PROGRAM PRG_Machine
VAR
	
	//empty recipe
	empty_recipe				:recipe;
	
	//debug
	after_debug_state					:INT :=0;

	
	Pusher :FB_Pusher;
	Compress: FB_Compress;
	Shield: FB_Shield;

	ZenonStart: NT_StartProcess;

	
	debug_counter: INT;
	tickcounter: INT;
	tickcounter2: INT;

	State: INT:= 0;
	state_old: INT:=0;
	StateNext: INT:= 0;
	
	SM_StepRequest: BOOL:=FALSE;
	singleStep: BOOL:=FALSE;
		
	Clamp_Security_Time: TIME := T#30S;
	ClampTimer: TON;
	//DwellTimer: TON;
	//SaveTickCounter: INT := 0;

	DatumTaught: BOOL;

	

	
	//stage
	stage_sh_push						:INT:=1;
	
END_VAR

VAR_OUTPUT

	rec_old		:recipe;
END_VAR

IF TRUE THEN
	debug_counter := debug_counter+1;
END_IF



qbCompressServoTorqueLimit := 1000;
qbPusherServoTorqueLimit := 1000;
qbShieldServoTorqueLimit := 1000;


//The state-machine
CASE State OF
	
0: //Copy config .txt file into machine settings
	


	//Zenon start process function call - appears to never generate errors
	
	//IF ZenonStart.Busy=FALSE THEN
	ZenonStart (
		NETID :=,
		//PATHSTR := 'Hard Disk\CP6606_Runtime\zenonRCE.exe', //'C:\PROGRAM Files\COPA-DATA\zenon 7.20 SP0\Zenrt32.exe',
		//DIRNAME := 'Hard Disk\CP6606_Runtime',  //'C:\Program Files\COPA-DATA\zenon 7.20 SP0',
		PATHSTR := 'Hard Disk\ZenonRunTime\zenonRCE.exe', //'C:\PROGRAM Files\COPA-DATA\zenon 7.20 SP0\Zenrt32.exe',
		DIRNAME := 'Hard Disk\ZenonRunTime',  //'C:\Program Files\COPA-DATA\zenon 7.20 SP0',
		COMNDLINE := '',
		START := TRUE,
		TMOUT := DEFAULT_ADS_TIMEOUT
		);
	StateNext := 10;



10: 
	qxEnableE_Stop := FALSE;
	tickcounter := 0;
	StateNext := 15;

15: //Check E-Stop relay is not set then Enable and initialise stuff - disable drive to clear errors

	

	//IF ixCabinetE_StopButtonOkay THEN
	qxEnableE_Stop := TRUE;
	StateNext := 20;
	//ELSE
	//	ResetLampController.State := SlowFlash;
	//END_IF
	
20: // Look for E-Stop button reset
	IF ixCabinetE_StopButtonOkay THEN
		//ResetLampController.State := steady;
		StateNext := 30;
	ELSE
		 
		ResetLampController.State := SlowFlash;
			
	END_IF
	
	//here
30: // Wait for operator to hit reset button
	
	IF ixE_StopRelayOkay THEN
		ResetLampController.State := off;
		StateNext := 40;
		tickcounter := 0;
	ELSE
		ResetLampController.State := steady;
		


	END_IF

40: // look for guard closed - disable drive to clear errors
	//sSystemStateMed := F_DisplayText("Guard Open",0);	
	//CurrentProcessState	:= F_DisplayText("not ready",0);	//Main Screen	

	
	IF NOT ixGuardOkay THEN
		ResetLampController.State := FastFlash;		
	ELSE
		ResetLampController.State := off;
		//sSystemStateMed := F_DisplayText("Initialising Axes",0);	
		tickcounter := 0;
		StateNext := 50;
	END_IF

50:
	IF ixGuardRelayOkay THEN
		statenext:=100;
	END_IF
	
100: // wait 2 scans for power supply to drive to stabilise
	tickcounter := tickcounter + 1;
	IF tickcounter >= 2 THEN
		tickcounter := 0;
		StateNext := 105;
	END_IF

105:
	IF NOT ixresetbutton THEN
		statenext:=110;
	END_IF	
	
110: // prepare for Servo motion - enable drive
//you are here!!!!!!!!!!!!!!!!!!!!!!!!!!!!
	//IF NOT ixResetButton THEN
		
		
	
	Shield._Enable();
	Pusher._Enable();
	Compress._Enable();
		
	tickcounter := tickcounter + 1;
	IF tickcounter >= 100 THEN
		tickcounter := 0;

		StateNext := 115;
	END_IF	
	//END_IF


	
115: 
	
	//IF Shield.HomeExecuted = FALSE OR Pusher.HomeExecuted = FALSE OR Compress.HomeExecuted = FALSE THEN
	IF language.english THEN
		Stage_Name := 'Beginning';
	ELSE
		Stage_Name := 'Início';
	END_IF
	Maintenance_Visibility:=TRUE;
	qxStartButtonLamp:=TRUE;
	IF (ixStartButton OR Step_Next OR ixStart_Button_Machine) THEN
		IF (parameter_violation = FALSE) THEN
			qxStartButtonLamp:=FALSE;
			StateNext := 116;
			Step_Next := FALSE;
			Clamp_Alarm:=FALSE;
			Maintenance_Visibility:=FALSE;
			stage_sh_push:=1;
			//Stage_Name := 'Homing and Offsetting';



		ELSE
			Step_Next:=FALSE;
		END_IF
	END_IF

	
116:
	IF (NOT ixstartbutton) AND NOT ixstart_button_machine THEN
		//general_offset_update();

		
		statenext:=117;
	END_IF
	
117:
	IF Compress.HomeExecuted=TRUE AND 
	   Shield.HomeExecuted = TRUE AND 
	   Pusher.HomeExecuted = TRUE AND
	   Pusher.OffsetExecuted = TRUE AND
	   Shield.OffsetExecuted = TRUE AND
	   Compress.OffsetExecuted = TRUE AND
	   Debug_Mode = FALSE THEN
	   
	   statenext:= 130;
	ELSE
		statenext:=120;
	END_IF
	
	Shield.Shield_param:=recipe_screen;
	Compress.Compress_Param := recipe_screen;
	Pusher.Pusher_Param := recipe_screen;
	//ELSE
	//	StateNext:=129;
	//	after_debug_state:=128;
	//END_IF
		
120: //you are here!!!!!!!!!!!!

	IF language.english THEN
		Stage_Name := 'Homing';
	ELSE
		Stage_Name := 'Ir para Início';
	END_IF
	IF Pusher.HomeExecuted = FALSE THEN 
		Pusher._Home();
	END_IF
	
	IF Compress.HomeExecuted = FALSE THEN
		Compress._Home();
	END_IF
	
	
	IF Compress.HomeExecuted AND Pusher.HomeExecuted THEN
		StateNext := 125;                //directly to end
		//Compress.HomeExecuted:=FALSE;
		//Pusher.HomeExecuted:=FALSE;
		
	END_IF
	
125:
	//random:='arda';
	IF Shield.HomeExecuted = FALSE THEN
		Shield._Home();
		
	ELSE
		StateNext := 129;
		IF language.english THEN
			Stage_Name := 'Homing done';
		ELSE
			Stage_Name := 'Ir para início concluído';
		END_IF
		after_debug_state :=127;
		//Shield.HomeExecuted := FALSE;
	END_IF

127:
	
	IF language.english THEN	
		Stage_Name := 'Offsetting';
	ELSE
		Stage_Name := 'Desviando';
	END_IF
	
	IF Compress.OffsetExecuted = FALSE THEN
		Compress.Offset(enable:=TRUE);
	END_IF
	
	IF Shield.OffsetExecuted = FALSE THEN
		Shield.Offset(enable:=TRUE);
	END_IF
	
	IF Pusher.OffsetExecuted = FALSE THEN
		Pusher.Offset(enable:=TRUE);
	END_IF
	
	IF Pusher.OffsetExecuted AND Shield.OffsetExecuted AND Compress.OffsetExecuted THEN
		Pusher.Offset(enable:=FALSE);
		Shield.Offset(enable:=FALSE);
		Compress.Offset(enable:=FALSE);
		
		rec_old:=Shield.Shield_Param;     //old values
		
		IF language.english THEN
			Stage_Name := 'Offsetting done';
		ELSE
			Stage_Name :='Desvio concluído';	
		END_IF
		
		Maintenance_Visibility := TRUE;
		qxStartButtonLamp:=TRUE;
		IF (ixStartButton OR Step_Next OR ixStart_Button_Machine) THEN
			IF (parameter_violation =FALSE) THEN
				qxStartButtonLamp:=FALSE;
				
				Shield.Shield_param:=recipe_screen;
				Compress.Compress_Param := recipe_screen;
				Pusher.Pusher_Param := recipe_screen;
			
				StateNext:=128;
				Step_Next:=FALSE;
				Maintenance_Visibility := FALSE;
			ELSE
				Step_Next:=FALSE;
			END_IF
		END_IF
	END_IF
	
128:	
	IF NOT ixstartbutton AND NOT ixstart_button_machine THEN
		statenext:=130;
	END_IF	

129: //debug	
	
	IF _debug(enable:=TRUE) THEN
		_debug(enable:=FALSE);
		statenext:=131;
	END_IF
		
130: //stage 1

	//IF ixstartbutton AND NOT ixstart_button_machine THEN
	IF language.english THEN
		Stage_Name := 'Compress Tobacco';
	ELSE
		Stage_Name := 'Comprimir Tabaco';
	END_IF
	
	IF qxClamp = FALSE THEN
		qxClamp:=TRUE;
		ClampTimer.IN:=TRUE;
		ClampTimer.PT:=Clamp_Security_Time;

	END_IF
	
	//IF Compress.Stage1Executed = FALSE THEN

	Compress._compress_tobacco(Enable:=TRUE);
	Compress.HomeExecuted:=FALSE;	
	
	IF Compress.axis_ready THEN	//Compress.Stage1Executed := FALSE;
		StateNext := 129;
		after_debug_state:=135;
		Compress._compress_tobacco(Enable:=FALSE);
		
		
		IF language.english THEN
			Stage_Name := 'Compress Tobacco done';
		ELSE
			Stage_Name := 'Comprimir tabaco concluído';
		END_IF
		
	END_IF
	//END_IF

131: //after_each_debug
	IF NOT ixStartButton AND NOT ixStart_Button_Machine THEN
	
		statenext:=after_debug_state;
	END_IF
135://stage2
	
	IF language.english THEN
		Stage_Name := concat('Shield-Pusher Stage ',INT_TO_STRING(stage_sh_push));
	ELSE
		Stage_Name := concat('Empurrador-proteção Estágio',INT_TO_STRING(stage_sh_push));
	END_IF
	
	Pusher.HomeExecuted:=FALSE;
	Shield.HomeExecuted:=FALSE;
		
	Pusher._absolute_move(Enable:=TRUE,Stage:=stage_sh_push);
	Shield._absolute_move(Enable:=TRUE,Stage:=stage_sh_push);
	IF pusher.axis_ready AND shield.axis_ready THEN	
		Statenext:= 129;
		IF stage_sh_push =6 THEN
			after_debug_state := 150;
			stage_sh_push:=0;
		ELSE
			after_debug_state := 135;
		END_IF
		Pusher._absolute_move(Enable:=FALSE,Stage:=stage_sh_push);
		Shield._absolute_move(Enable:=FALSE,Stage:=stage_sh_push);
		stage_sh_push:=stage_sh_push+1;
		
		IF language.english THEN
			Stage_Name:=concat(Stage_Name,' done');
		ELSE
			Stage_Name:=concat(Stage_Name,' concluído');
		END_IF
	END_IF	
	


150: //stage 5
	IF language.english THEN
		Stage_Name := 'Retract all';
	ELSE
		Stage_Name := 'Retrair tudo';
	END_IF
	//IF 	Shield._retract(Enable:=TRUE) AND Pusher._retract(Enable:=TRUE) AND Compress._retract(Enable:=TRRUE) THEN
	Pusher._Retract(enable:=TRUE);
	Shield._retract(enable:=TRUE);
	Compress._retract(enable:=TRUE);

	IF Compress.axis_ready AND Shield.Axis_ready AND Pusher.axis_ready THEN
		Pusher._Retract(enable:=FALSE);
		Shield._retract(enable:=FALSE);
		Compress._retract(enable:=FALSE);
		Statenext:=290;
		
		IF language.english THEN
			Stage_Name := 'Retract All Done';
		ELSE
			Stage_Name := 'Retrair tudo concluído';
		END_IF
	END_IF	

290:
	product_count:=product_count+1;
	statenext:=300;


300: //end
	
	Pusher.HomeExecuted:= TRUE;
	Shield.HomeExecuted:=TRUE;
	Compress.HomeExecuted:=TRUE;
	statenext:= 115;

	
1000: // overtorque
	
	//StartLoad := FALSE;
	
	tickcounter:=0;
	
	qxclamp:=FALSE;
	ClampTimer.IN:=FALSE;
	ClampTimer.PT:=Clamp_Security_Time;
	
	IF Pusher.PusherServo.xstopped AND Shield.ShieldServo.xstopped AND Compress.CompressServo.xstopped THEN
		Pusher._Reset();
		Shield._Reset();
		Compress._Reset();
		Statenext:=1005;
	END_IF

1005:
	
	IF tickcounter >1000 THEN
		statenext:=2000;
		tickcounter:=0;
	ELSE
		tickcounter:=tickcounter+1;
	END_IF

	
2000: // estop //overtorque
	
	tickcounter:= tickcounter+1;
	IF	tickcounter = 100 THEN
		tickcounter:=0;
		
		statenext:=15;
		overtorque_alarm:=FALSE;
	END_IF

2001: //guard
	tickcounter:= tickcounter+1;
	IF	tickcounter = 100 THEN
		tickcounter:=0;
		
		statenext:= 40;
		
	END_IF

2010: // clamp alarm
	
	tickcounter:= tickcounter+1;

	
	IF clamp_alarm THEN
		
		IF	tickcounter = 3000 THEN
			tickcounter:=0;
			statenext:=100;
			Clamp_Cooling := FALSE;
			Clamp_Alarm := FALSE;
		ELSE
			Clamp_Cooling := TRUE;
			
			IF Pusher.PusherServo.xstopped AND Shield.ShieldServo.xstopped AND Compress.CompressServo.xstopped THEN
				Pusher._Reset();
				Shield._Reset();
				Compress._Reset();
			END_IF
		END_IF
	END_IF 



2015://stop button
	tickcounter:= tickcounter+1;
	IF	tickcounter = 100 THEN
		tickcounter:=0;
		statenext:=100;
		
	ELSIF Pusher.PusherServo.xstopped AND Shield.ShieldServo.xstopped AND Compress.CompressServo.xstopped THEN
		Pusher._Reset();
		Shield._Reset();
		Compress._Reset();
		
	END_IF

2020: //force home

	IF shield.ShieldServo.xHalted AND pusher.pusherservo.xHalted AND compress.compressservo.xhalted THEN
		Pusher._soft_Reset();
		Shield._soft_Reset();
		Compress._soft_Reset();
		IF compress.offsetExecuted AND shield.Offsetexecuted AND pusher.offsetexecuted THEN
			statenext:=200;
		ELSE

			statenext:=210;
		END_IF
	END_IF

2030: //compress setting
	IF shield.ShieldServo.xHalted AND pusher.pusherservo.xHalted AND compress.compressservo.xhalted THEN
		Pusher._soft_Reset();
		Shield._soft_Reset();
		Compress._soft_Reset();
		
		
		Compress.HomeExecuted:=FALSE;
		Shield.HomeExecuted:=FALSE;
		Pusher.HomeExecuted:=FALSE;
	
		Compress.OffsetExecuted:=FALSE;
		Shield.OffsetExecuted:=FALSE;
		Pusher.OffsetExecuted:=FALSE;
		
		reset_rec_old();
		
		IF NOT compress_settings.done AND yellow_visibility.maintenance THEN
			statenext:=230;
		ELSE
			statenext:=115;
			compress_settings.done:=FALSE;
		END_IF
	END_IF


	
	
200:

	IF language.english THEN
		Stage_Name := 'Going to Home Position';	
	ELSE
		Stage_Name := 'Indo para Posição Inicial';
	END_IF
	
	
	
	Pusher._force_home(enable:=TRUE);
	
	IF tickcounter > 100 THEN
		Shield._force_home(enable:=TRUE);
	ELSE
		tickcounter:=tickcounter+1;
	END_IF
			
	Compress._force_home(enable:=TRUE);
	
	
	IF Compress.axis_ready AND Pusher.axis_ready AND Shield.Axis_ready THEN
		tickcounter:=0;
		Pusher._force_home(enable:=FALSE);
		Shield._force_home(enable:=FALSE);
		Compress._force_home(enable:=FALSE);
		Statenext:=300;
		
	END_IF

210:
	Compress.HomeExecuted:=FALSE;
	Shield.HomeExecuted:=FALSE;
	Pusher.HomeExecuted:=FALSE;
	
	Compress.OffsetExecuted:=FALSE;
	Shield.OffsetExecuted:=FALSE;
	Pusher.OffsetExecuted:=FALSE;
	
	Shield.Shield_param:=recipe_screen;
	Compress.Compress_Param := recipe_screen;
	Pusher.Pusher_Param := recipe_screen;
	
	reset_rec_old();
	
	Statenext:=211;

211:

	IF language.english THEN
		Stage_Name := 'Going to Home Position';	
	ELSE
		Stage_Name := 'Indo para Posição Inicial';
	END_IF
	
	IF Pusher.HomeExecuted = FALSE THEN 
		Pusher._Home();
		
	END_IF
	
	IF Compress.HomeExecuted = FALSE THEN
		Compress._Home();
		
	END_IF
	
	IF shield.HomeExecuted = FALSE THEN
		IF tickcounter>100 THEN
			Shield._Home();
		ELSE
			tickcounter:=tickcounter+1;
		END_IF
	END_IF
	
	IF Compress.HomeExecuted AND Pusher.HomeExecuted AND Shield.HomeExecuted THEN
		StateNext := 212;
		tickcounter:=0;                
		
	END_IF
	

212:

	IF Compress.OffsetExecuted = FALSE THEN
		Compress.Offset(enable:=TRUE);
	END_IF
	
	IF Shield.OffsetExecuted = FALSE THEN
		Shield.Offset(enable:=TRUE);
	END_IF
	
	IF Pusher.OffsetExecuted = FALSE THEN
		Pusher.Offset(enable:=TRUE);
	END_IF
	
	IF Pusher.OffsetExecuted AND Shield.OffsetExecuted AND Compress.OffsetExecuted THEN
		Pusher.Offset(enable:=FALSE);
		Shield.Offset(enable:=FALSE);
		Compress.Offset(enable:=FALSE);
		rec_old:= shield.Shield_Param;
		statenext:=300;
	END_IF

230:
	Compress._manuel(TRUE);
	
	IF compress_settings.find THEN
		statenext:=235;
		compress_settings.old_distance:=compress.compressservo.fActualPosition;
		Compress._manuel(FALSE);	
	END_IF
	
	IF compress_settings.done OR NOT yellow_visibility.maintenance THEN
		statenext:=2030;
		Compress._manuel(FALSE);
		compress_settings.distance_vis:=FALSE;
		//compress_settings.done:=FALSE;
		Compress._Halt();
		Shield._Halt();
		Pusher._Halt();
		
	END_IF
	
235://here
	Compress._Home_without_resetting(TRUE);
	compress_settings.distance_vis:=FALSE;
	
	IF Compress.axis_ready THEN
		Compress_settings.distance := Compress_settings.old_distance - compress.compressservo.fActualPosition;
		StateNext:=230;
		compress_settings.distance_vis:=TRUE;
		Compress._Home_without_resetting(FALSE);
	END_IF
	
	IF compress_settings.done OR NOT yellow_visibility.maintenance THEN
		statenext:=2030;
		Compress._Home_without_resetting(FALSE);
		compress_settings.distance_vis:=FALSE;
		//compress_settings.done:=FALSE;
		Compress._Halt();
		Shield._Halt();
		Pusher._Halt();
		
		
	END_IF


	
END_CASE

Pusher._Update();
Shield._Update();
Compress._Update();
ClampTimer();

axis_offset_or_not();

//maintenance visibility and stop button light
start_lamp_control();

//Motor Overtorque
motor_overtorque();



//Toggole Clamp
funct_toggle_clamp();

//Home
funct_force_home();

//stop button
funct_stop();

//Clamp Err
funct_clamp_err();

//compress setting
funct_compress_setting();


//guard
funct_guard_open();


//estop
funct_e_stop();

//IF State <> StateNext THEN - step through the state machine if required
coder_debug();

METHOD _debug : BOOL
VAR_INPUT
	enable				:BOOL;
END_VAR
IF enable THEN
	
	IF Debug_Mode THEN
		Maintenance_Visibility := TRUE;
		qxStartButtonLamp:=TRUE;
		IF (ixStartButton OR Step_Next OR ixStart_Button_Machine) THEN
			IF Parameter_Violation = FALSE THEN
				
				Step_Next:=FALSE;
				
				_debug:=TRUE;
				
				Maintenance_Visibility := FALSE;
				qxStartButtonLamp:=FALSE;
			
				Shield.Shield_param:=recipe_screen;
				Compress.Compress_Param := recipe_screen;
				Pusher.Pusher_Param := recipe_screen;
			ELSE
				Step_Next:=FALSE;
			END_IF
		END_IF
	ELSE
		//StateNext:=130;
		_debug:=TRUE;
		Maintenance_Visibility := FALSE;
	END_IF
	
	
ELSE
	_debug:=FALSE;
END_IF
END_METHOD

METHOD axis_offset_or_not : BOOL
VAR_INPUT
END_VAR
	//rec_old:=Shield.Shield_Param;     //old values

	
	//Shield.Shield_param:=recipe_screen;         //new valuses
	//Compress.Compress_Param := recipe_screen;
	//Pusher.Pusher_Param := recipe_screen;
	
IF statenext<>127 AND statenext<> 212 THEN
	IF rec_old.other.Shield_Home_Offset <> recipe_screen.Other.Shield_Home_Offset THEN

		Shield.OffsetExecuted:=FALSE;
	END_IF
	
	IF rec_old.other.Pusher_Home_Offset <> recipe_screen.Other.Pusher_Home_Offset THEN
		Pusher.OffsetExecuted:=FALSE;
	END_IF
	
	IF rec_old.other.Compress_Home_Offset <> recipe_screen.Other.Compress_Home_Offset THEN
		Compress.OffsetExecuted:=FALSE;
	END_IF
END_IF
END_METHOD

METHOD coder_debug : BOOL
VAR_INPUT
END_VAR
IF singleStep AND statenext > 119 THEN
	//IF NOT SM_StepRequest THEN
	//	SM_StepRequest := TRUE; 
	//END_IF
	IF SM_StepRequest THEN
		SM_StepRequest := FALSE;
		State := StateNext;
	END_IF
ELSE
	State := StateNext;
END_IF
END_METHOD

METHOD funct_clamp_err : BOOL
VAR_INPUT
END_VAR
IF (Clamptimer.Q=TRUE) AND StateNext >= 100 AND StateNext <= 300 THEN 
	
	tickcounter:=0;
	//Message:='Clamp Overtime';
	qxClamp:=FALSE;

	
	ClampTimer.IN:=FALSE;
	ClampTimer.PT:=Clamp_Security_Time;
	
	Clamp_Alarm:=TRUE;
	
	Compress._mc_stop();
	Shield._mc_stop();
	Pusher._mc_stop();
	StateNext := 2010;

END_IF
END_METHOD

METHOD funct_compress_setting : BOOL
VAR_INPUT
END_VAR
IF compress_settings.button AND StateNext >= 115 AND StateNext <= 300 THEN
	compress_settings.button:=FALSE;
	
	IF statenext < 230 OR statenext >250 THEN
		StateNext := 2030;
		tickcounter:=0;
	
		compress_settings.done:=FALSE;
	
	
		qxclamp:=FALSE;
		ClampTimer.IN:=FALSE;
		ClampTimer.PT:=Clamp_Security_Time;
	
		shield._Halt();
		pusher._Halt();
		compress._Halt();
	END_IF
	
ELSE
	compress_settings.button:=FALSE;
END_IF
END_METHOD

METHOD funct_e_stop : BOOL
VAR_INPUT
END_VAR
IF (NOT ixCabinetE_StopButtonOkay) AND StateNext >= 30 AND StateNext <= 300 THEN 
	
	tickcounter:=0;
	
	//Message:='E-stop Pressed';
	
	qxclamp:=FALSE;
	ClampTimer.IN:=FALSE;
	ClampTimer.PT:=Clamp_Security_Time;
	

	
	//IF Compress.CompressServo.xStopped AND Shield.ShieldServo.xStopped AND Pusher.PusherServo.xStopped THEN
	StateNext := 2000;
	Pusher._Reset();
	Shield._Reset();
	Compress._Reset();
	//END_IF
END_IF
END_METHOD

METHOD funct_force_home : BOOL
VAR_INPUT
END_VAR
IF (Force_Home) AND StateNext >= 115 AND StateNext <= 300 THEN 
	Force_Home:=FALSE;
	
	IF statenext < 200 OR statenext >220 THEN
		StateNext := 2020;
		tickcounter:=0;
	
	
	
	
		qxclamp:=FALSE;
		ClampTimer.IN:=FALSE;
		ClampTimer.PT:=Clamp_Security_Time;
	
		shield._Halt();
		pusher._Halt();
		compress._Halt();
	END_IF

END_IF
END_METHOD

METHOD funct_guard_open : BOOL
VAR_INPUT
END_VAR
IF (NOT ixGuardRelayOkay) AND StateNext >= 50 AND StateNext <= 300 THEN 
	
	StateNext := 2001;
	tickcounter:=0;
	
	//Message:='Guard Open';
	
	qxclamp:=FALSE;
	ClampTimer.IN:=FALSE;
	ClampTimer.PT:=Clamp_Security_Time;
	
	IF Pusher.HomeExecuted= FALSE OR Shield.HomeExecuted = FALSE OR Compress.HomeExecuted = FALSE THEN
		Pusher._Reset();
		Shield._Reset();
		Compress._Reset();
	ELSE
		Pusher._Reset_Medium();
		Shield._Reset_Medium();
		Compress._Reset_Medium();
	END_IF
END_IF
END_METHOD

METHOD funct_stop : BOOL
VAR_INPUT
END_VAR
IF NOT ixstop_button AND (Statenext<>151) AND StateNext >= 100 AND StateNext <= 300 THEN
	//	state_old:=statenext;
	//	statenext:= 151;
	tickcounter:=0;
	//Message:='Clamp Overtime';
	qxClamp:=FALSE;

	
	ClampTimer.IN:=FALSE;
	ClampTimer.PT:=Clamp_Security_Time;
	
	
	
	Compress._mc_stop();
	Shield._mc_stop();
	Pusher._mc_stop();
	StateNext := 2015;
	
	
END_IF
END_METHOD

METHOD funct_toggle_clamp : BOOL
VAR_INPUT
END_VAR
IF StateNext >= 115 AND StateNext <= 300 AND Toggle_Clamp THEN
	Toggle_Clamp := FALSE;
	IF qxClamp = FALSE THEN
		
		qxClamp:=TRUE;
		ClampTimer.IN:=TRUE;
		ClampTimer.PT:=Clamp_Security_Time;

	ELSE
		
		qxClamp:=FALSE;
		ClampTimer.IN:=FALSE;
		ClampTimer.PT:=Clamp_Security_Time;
		
	END_IF
	
	
END_IF
END_METHOD

METHOD motor_overtorque : BOOL
VAR
	torque_lim			:LREAL;
	current_torque_shield		:LREAL;
	current_torque_compress		:LREAL;
	current_torque_pusher		:LREAL;
	
END_VAR
IF StateNext >= 110 AND StateNext <= 300  THEN					// machine is running
	
	torque_lim:=limits_screen.max_torque;
	//torque_lim:=2000;
	
	current_torque_shield:=ibshieldservotorque;
	current_torque_pusher:=ibpusherservotorque;
	current_torque_compress:=ibcompressservotorque;
	
	IF current_torque_compress  > torque_lim OR current_torque_compress  < (-1*torque_lim) THEN					
		//Message := WSTRING_TO_STRING("Tobacco Compress Servo over-torque");
		StateNext := 1000;
		tickcounter:=0;
		overtorque_alarm:= TRUE;

		compress._mc_stop();
		shield._mc_stop();
		pusher._mc_stop();	
	END_IF
	
	IF current_torque_pusher  > torque_lim OR current_torque_pusher  < (-1*torque_lim) THEN						
		//Message := WSTRING_TO_STRING("Rod Pusher Servo over-torque");
		StateNext := 1000;
		tickcounter:=0;
		overtorque_alarm:= TRUE;
		
		compress._mc_stop();
		shield._mc_stop();
		pusher._mc_stop();	
			
	END_IF
	
	IF current_torque_shield  > torque_lim OR current_torque_shield  < (-1*torque_lim) THEN						
		//Message := WSTRING_TO_STRING("Rod Shield Servo over-torque");
		StateNext := 1000;
		tickcounter:=0;
		overtorque_alarm:= TRUE;

		compress._mc_stop();
		shield._mc_stop();
		pusher._mc_stop();		
	END_IF
END_IF
END_METHOD

METHOD reset_rec_old : BOOL
VAR_INPUT
END_VAR
rec_old:=empty_recipe;
END_METHOD

METHOD start_lamp_control : BOOL
VAR_INPUT
END_VAR
//IF 	StateNext <> 115 AND 
//	StateNext <> 127 THEN
//	qxStartButtonLamp:=FALSE;
//END_IF

IF 	StateNext <> 115 AND StateNext <> 127 AND StateNext <> 129 THEN
	qxStartButtonLamp:=FALSE;
	Maintenance_Visibility := FALSE;
END_IF
END_METHOD

METHOD StopClampTimer
VAR_INPUT
END_VAR
ClampTimer.IN:=FALSE;
ClampTimer.PT:= Clamp_Security_Time;
END_METHOD

END_PROGRAM

(* stored: Version 1.1.0.1, ProductVersion 3.1.4022.9
   POU PRG_Machine: Id {4059ff51-9b15-4d7b-8b65-432c3cf02eab}, SpecialFunc None
   Method _debug: Id {f6433566-6785-4878-8f43-678526334943}
   Method axis_offset_or_not: Id {d164c1fe-0cb6-4c44-9acc-255c3243d05d}
   Method coder_debug: Id {cb589c93-1c5f-40bc-8bd3-5a0a214df7d7}
   Method funct_clamp_err: Id {0531b7a1-3269-4dd0-aaf5-d310f7ea000a}
   Method funct_compress_setting: Id {13d31d39-a0f1-42cf-b0af-9bd86fb48dec}
   Method funct_e_stop: Id {4ccb4d2f-960e-4196-8bdd-1b13290cadda}
   Method funct_force_home: Id {157a9dae-2c6e-4248-bca1-03befd179033}
   Method funct_guard_open: Id {6038006e-bd91-43a7-ac1a-d5f8f2fbf802}
   Method funct_stop: Id {523098cb-cbef-4171-9dd6-3a588f471015}
   Method funct_toggle_clamp: Id {5b9d45e8-6c4a-48e8-a6de-c92875096aa8}
   Method motor_overtorque: Id {48735565-c2d5-4500-892e-2ffb096c9465}
   Method reset_rec_old: Id {44203f13-db00-491a-9168-cd6f7805302c}
   Method start_lamp_control: Id {3f09c7f5-6d41-4dbc-b351-ef97ecafa1ab}
   Method StopClampTimer: Id {d74d2087-e1fa-4163-bf2f-94ebc8b0fc77} *)
